# EPICS substitutions: watlowPMApp/Db/Watlow_PM_IOC_Alarm.substitutions
file Watlow_PM_IOC_Alarms.template
{
pattern
{PREFIX}
{"XF:07BM-ES{Watlow:1}"}
}

file save_restoreStatus.db
{
pattern {P}
        {"XF:07BM-ES{Watlow:1}"}
}

file ioc_sns.db
{
pattern {IOCNAME}
        {"XF:07BM-ES{Watlow:1}"}
}
